// TIA Portal V17 export
// export: Created 2021-12-03T08:13:13.0262068Z, ExportSetting WithDefaults, DisplayName Totally Integrated Automation Portal, DisplayVersion V17, DisplayName TIA Portal Openness, DisplayVersion V17, DisplayName TIA Portal Version Control Interface, DisplayVersion V17, DisplayName STEP 7 Professional, DisplayVersion V17, DisplayName STEP 7 Safety, DisplayVersion V17, DisplayName WinCC Advanced, DisplayVersion V17
DATA_BLOCK "FGDB_Safety_Perimeter"   // DB300, F_DB
VERSION : 0.1
// stored: AutoNumber false
   VAR
      RdyOpn : Bool;   // Готовность к открытию
      SAreaClose : Bool;   // Периметр безопасности закрыт
      SPBreak : Bool;   // Нелегальное открытие периметра
      RdyCls_P3 : Bool;   // Готовность к закрытию
      AckCls : Bool;   // Запрос на закрытие
      Opn : Bool;   // Происходит открытие
   END_VAR
BEGIN
END_DATA_BLOCK
